ABB RAPID module: prog-1.rapid

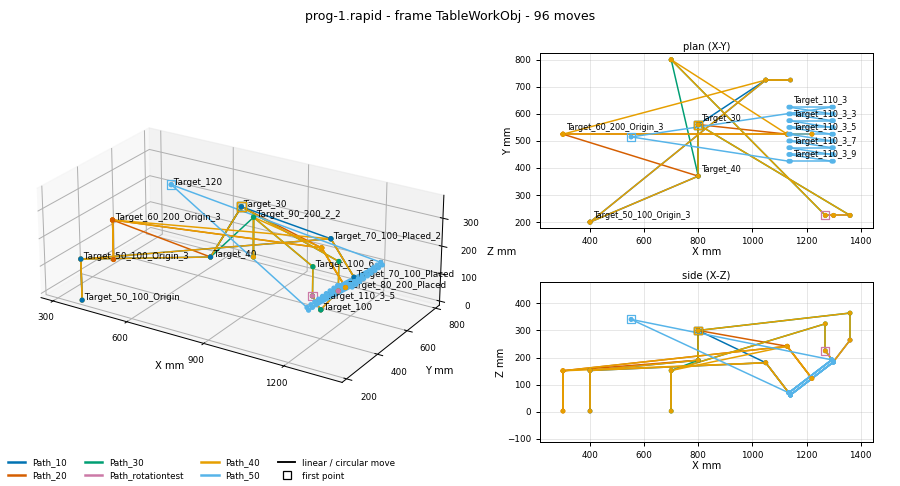
[picture p0: tool path of prog-1.rapid in frame TableWorkObj, 96 of 96 moves have a stored position in this frame; points joined in program order, loops and branches not executed]
MODULE Module1
    CONST robtarget Target_30:=[[800,560.525588833,300],[0.353553391,-0.612372436,0.612372436,0.353553391],[-1,0,-1,0],[9E+09,9E+09,9E+09,9E+09,9E+09,9E+09]];
    CONST robtarget Target_40:=[[800,370.00032529,189.999990631],[-0.000000004,-0.707106781,0.707106781,-0.000000004],[-1,0,-1,0],[9E+09,9E+09,9E+09,9E+09,9E+09,9E+09]];
    CONST robtarget Target_50_100_Origin_3:=[[400,199.9999982,152],[0.000000006,1,0,0],[0,0,-1,0],[9E+09,9E+09,9E+09,9E+09,9E+09,9E+09]];
    CONST robtarget Target_50_100_Origin:=[[400,200,2],[-0.000000006,1,0,0],[0,-1,-1,0],[9E+09,9E+09,9E+09,9E+09,9E+09,9E+09]];
    CONST robtarget Target_70_100_Placed_2:=[[1049.406562207,725,180.67251142],[-0.000000006,1,0,0],[-1,0,-2,0],[9E+09,9E+09,9E+09,9E+09,9E+09,9E+09]];
    CONST robtarget Target_70_100_Placed:=[[1140.720642254,725,61.669407321],[0,0.946930311,0,0.321438931],[-1,-1,-2,0],[9E+09,9E+09,9E+09,9E+09,9E+09,9E+09]];
    CONST robtarget Target_60_200_Origin_3:=[[300.000000926,524.99999882,151],[0.000000003,0.965925826,-0.258819045,-0.000000004],[0,0,-1,0],[9E+09,9E+09,9E+09,9E+09,9E+09,9E+09]];
    CONST robtarget Target_60_200_Origin:=[[300,525,2],[0,0.965925826,-0.258819045,0],[0,0,-1,0],[9E+09,9E+09,9E+09,9E+09,9E+09,9E+09]];
    CONST robtarget Target_80_200_Placed_2:=[[1128.741964994,525,241.548561714],[-0.000000006,1,0,0],[-1,0,-2,0],[9E+09,9E+09,9E+09,9E+09,9E+09,9E+09]];
    CONST robtarget Target_80_200_Placed:=[[1220.056045041,525,122.545460615],[0,0.946930311,0,0.321438931],[-1,-1,-2,0],[9E+09,9E+09,9E+09,9E+09,9E+09,9E+09]];
    CONST robtarget Target_90_200_2_2:=[[700,800,152],[0,0.965925826,0.258819045,0],[0,0,-2,0],[9E+09,9E+09,9E+09,9E+09,9E+09,9E+09]];
    CONST robtarget Target_90_200_2:=[[700,800,2],[0,0.965925826,0.258819045,0],[0,0,-2,0],[9E+09,9E+09,9E+09,9E+09,9E+09,9E+09]];
    CONST robtarget Target_100_6_2:=[[1269.56192856,225,324.667667022],[0.000000006,1,0,0],[-1,-1,-2,0],[9E+09,9E+09,9E+09,9E+09,9E+09,9E+09]];
    CONST robtarget Target_100_6:=[[1269.56192856,225,224.667667022],[0,0.94693013,0,0.321439465],[-1,-1,-2,0],[9E+09,9E+09,9E+09,9E+09,9E+09,9E+09]];
    CONST robtarget Target_100:=[[1300,225,185],[0,0.946930129,0,0.321439465],[-1,-1,-2,0],[9E+09,9E+09,9E+09,9E+09,9E+09,9E+09]];
    CONST robtarget Target_100_3:=[[1300,225,185],[0,0.946930129,0,-0.321439465],[-1,0,-2,0],[9E+09,9E+09,9E+09,9E+09,9E+09,9E+09]];
    CONST robtarget Target_100_3_2:=[[1360.876142881,225,264.335334045],[0,0.94693013,0,-0.321439465],[-1,0,-2,0],[9E+09,9E+09,9E+09,9E+09,9E+09,9E+09]];
    CONST robtarget Target_100_3_2_2:=[[1360.876142881,225,364.335334045],[0.000000006,1,0,0],[-1,-1,-2,0],[9E+09,9E+09,9E+09,9E+09,9E+09,9E+09]];
    CONST robtarget Target_110_2_10:=[[1293.303842438,625,191.355054252],[0.946930311,0,-0.321438931,0],[-1,-4,2,1],[9E+09,9E+09,9E+09,9E+09,9E+09,9E+09]];
    CONST robtarget Target_110_2:=[[1299.391447774,625,183.421513979],[0.946930311,0,-0.321438931,0],[-1,-4,2,1],[9E+09,9E+09,9E+09,9E+09,9E+09,9E+09]];
    CONST robtarget Target_110_3:=[[1140.720642308,625,61.669407251],[0.946930311,0,-0.321438931,0],[-1,-4,2,1],[9E+09,9E+09,9E+09,9E+09,9E+09,9E+09]];
    CONST robtarget Target_110_3_10:=[[1134.633036972,625,69.602947524],[0.946930311,0,-0.321438931,0],[-1,-4,2,1],[9E+09,9E+09,9E+09,9E+09,9E+09,9E+09]];
    CONST robtarget Target_110_2_2_2:=[[1293.303842438,600,191.355054252],[0.946930311,0,-0.321438931,0],[-1,-4,2,1],[9E+09,9E+09,9E+09,9E+09,9E+09,9E+09]];
    CONST robtarget Target_110_2_2:=[[1299.391447774,600,183.421513979],[0.946930311,0,-0.321438931,0],[-1,-4,2,1],[9E+09,9E+09,9E+09,9E+09,9E+09,9E+09]];
    CONST robtarget Target_110_3_2:=[[1140.720642308,600,61.669407251],[0.946930311,0,-0.321438931,0],[-1,-4,2,1],[9E+09,9E+09,9E+09,9E+09,9E+09,9E+09]];
    CONST robtarget Target_110_3_2_2:=[[1134.633036972,600,69.602947524],[0.946930311,0,-0.321438931,0],[-1,-4,2,1],[9E+09,9E+09,9E+09,9E+09,9E+09,9E+09]];
    CONST robtarget Target_110_2_3_2:=[[1293.303842438,575,191.355054252],[0.946930311,0,-0.321438931,0],[-1,-4,2,1],[9E+09,9E+09,9E+09,9E+09,9E+09,9E+09]];
    CONST robtarget Target_110_2_3:=[[1299.391447774,575,183.421513979],[0.946930311,0,-0.321438931,0],[-1,-4,2,1],[9E+09,9E+09,9E+09,9E+09,9E+09,9E+09]];
    CONST robtarget Target_110_3_3:=[[1140.720642308,575,61.669407251],[0.946930311,0,-0.321438931,0],[-1,-4,2,1],[9E+09,9E+09,9E+09,9E+09,9E+09,9E+09]];
    CONST robtarget Target_110_3_3_2:=[[1134.633036972,575,69.602947524],[0.946930311,0,-0.321438931,0],[-1,-4,2,1],[9E+09,9E+09,9E+09,9E+09,9E+09,9E+09]];
    CONST robtarget Target_110_2_4_2:=[[1293.303842438,550,191.355054252],[0.946930311,0,-0.321438931,0],[-1,-4,2,1],[9E+09,9E+09,9E+09,9E+09,9E+09,9E+09]];
    CONST robtarget Target_110_2_4:=[[1299.391447774,550,183.421513979],[0.946930311,0,-0.321438931,0],[-1,-4,2,1],[9E+09,9E+09,9E+09,9E+09,9E+09,9E+09]];
    CONST robtarget Target_110_3_4:=[[1140.720642308,550,61.669407251],[0.946930311,0,-0.321438931,0],[-1,-4,2,1],[9E+09,9E+09,9E+09,9E+09,9E+09,9E+09]];
    CONST robtarget Target_110_3_4_2:=[[1134.633036972,550,69.602947524],[0.946930311,0,-0.321438931,0],[-1,-4,2,1],[9E+09,9E+09,9E+09,9E+09,9E+09,9E+09]];
    CONST robtarget Target_110_2_5_2:=[[1293.303842438,525,191.355054252],[0.946930311,0,-0.321438931,0],[-1,-4,2,1],[9E+09,9E+09,9E+09,9E+09,9E+09,9E+09]];
    CONST robtarget Target_110_2_5:=[[1299.391447774,525,183.421513979],[0.946930311,0,-0.321438931,0],[-1,-4,2,1],[9E+09,9E+09,9E+09,9E+09,9E+09,9E+09]];
    CONST robtarget Target_110_3_5:=[[1140.720642308,525,61.669407251],[0.946930311,0,-0.321438931,0],[-1,-4,2,1],[9E+09,9E+09,9E+09,9E+09,9E+09,9E+09]];
    CONST robtarget Target_110_3_5_2:=[[1134.633036972,525,69.602947524],[0.946930311,0,-0.321438931,0],[-1,-4,2,1],[9E+09,9E+09,9E+09,9E+09,9E+09,9E+09]];
    CONST robtarget Target_110_2_6_2:=[[1293.303842438,500,191.355054252],[0.946930311,0,-0.321438931,0],[-1,-4,2,1],[9E+09,9E+09,9E+09,9E+09,9E+09,9E+09]];
    CONST robtarget Target_110_2_6:=[[1299.391447774,500,183.421513979],[0.946930311,0,-0.321438931,0],[-1,-4,2,1],[9E+09,9E+09,9E+09,9E+09,9E+09,9E+09]];
    CONST robtarget Target_110_3_6:=[[1140.720642308,500,61.669407251],[0.946930311,0,-0.321438931,0],[-1,-4,2,1],[9E+09,9E+09,9E+09,9E+09,9E+09,9E+09]];
    CONST robtarget Target_110_3_6_2:=[[1134.633036972,500,69.602947524],[0.946930311,0,-0.321438931,0],[-1,-4,2,1],[9E+09,9E+09,9E+09,9E+09,9E+09,9E+09]];
    CONST robtarget Target_110_2_7_2:=[[1293.303842438,475,191.355054252],[0.946930311,0,-0.321438931,0],[-1,-4,2,1],[9E+09,9E+09,9E+09,9E+09,9E+09,9E+09]];
    CONST robtarget Target_110_2_7:=[[1299.391447774,475,183.421513979],[0.946930311,0,-0.321438931,0],[-1,-4,2,1],[9E+09,9E+09,9E+09,9E+09,9E+09,9E+09]];
    CONST robtarget Target_110_3_7:=[[1140.720642308,475,61.669407251],[0.946930311,0,-0.321438931,0],[-1,-4,2,1],[9E+09,9E+09,9E+09,9E+09,9E+09,9E+09]];
    CONST robtarget Target_110_3_7_2:=[[1134.633036972,475,69.602947524],[0.946930311,0,-0.321438931,0],[-1,-4,2,1],[9E+09,9E+09,9E+09,9E+09,9E+09,9E+09]];
    CONST robtarget Target_110_2_8_2:=[[1293.303842438,450,191.355054252],[0.946930311,0,-0.321438931,0],[-1,-4,2,1],[9E+09,9E+09,9E+09,9E+09,9E+09,9E+09]];
    CONST robtarget Target_110_2_8:=[[1299.391447774,450,183.421513979],[0.946930311,0,-0.321438931,0],[-1,-4,2,1],[9E+09,9E+09,9E+09,9E+09,9E+09,9E+09]];
    CONST robtarget Target_110_3_8:=[[1140.720642308,450,61.669407251],[0.946930311,0,-0.321438931,0],[-1,-4,2,1],[9E+09,9E+09,9E+09,9E+09,9E+09,9E+09]];
    CONST robtarget Target_110_3_8_2:=[[1134.633036972,450,69.602947524],[0.946930311,0,-0.321438931,0],[-1,-4,2,1],[9E+09,9E+09,9E+09,9E+09,9E+09,9E+09]];
    CONST robtarget Target_110_2_9_2:=[[1293.303842438,425,191.355054252],[0.946930311,0,-0.321438931,0],[-1,-4,2,1],[9E+09,9E+09,9E+09,9E+09,9E+09,9E+09]];
    CONST robtarget Target_110_2_9:=[[1299.391447774,425,183.421513979],[0.946930311,0,-0.321438931,0],[-1,-4,2,1],[9E+09,9E+09,9E+09,9E+09,9E+09,9E+09]];
    CONST robtarget Target_110_3_9:=[[1140.720642308,425,61.669407251],[0.946930311,0,-0.321438931,0],[-1,-4,2,1],[9E+09,9E+09,9E+09,9E+09,9E+09,9E+09]];
    CONST robtarget Target_110_3_9_2:=[[1134.633036972,425,69.602947524],[0.946930311,0,-0.321438931,0],[-1,-4,2,1],[9E+09,9E+09,9E+09,9E+09,9E+09,9E+09]];
    CONST robtarget Target_120:=[[552,514.814,340.825],[0.612372436,0.353553391,0.612372436,0.353553391],[0,-3,2,1],[9E+09,9E+09,9E+09,9E+09,9E+09,9E+09]];
    CONST robtarget Target_Patch200:=[[300,525,2],[0,0.965925826,-0.258819045,0],[0,0,-1,0],[9E+09,9E+09,9E+09,9E+09,9E+09,9E+09]];
!***********************************************************
    !
    ! Module:  Module1
    !
    ! Description:
    !   <Insert description here>
    !
    ! Author: tgell
    !
    ! Version: 1.0
    !
    !***********************************************************


    !***********************************************************
    !
    ! Procedure main
    !
    !   This is the entry point of your program
    !
    !***********************************************************
    PROC main()
        Path_20;
        Path_50;
        !Add your code here
    ENDPROC
    PROC Path_10()
        MoveL Target_30,v400,z100,Tooldata_1\WObj:=TableWorkObj;
        MoveL Target_40,v400,z100,Tooldata_1\WObj:=TableWorkObj;
        MoveL Target_50_100_Origin_3,v400,z100,Tooldata_1\WObj:=TableWorkObj;
        MoveL Target_50_100_Origin,v60,z100,Tooldata_1\WObj:=TableWorkObj;
        WaitTime 3;
        PulseDO att_100;
        MoveL Target_50_100_Origin_3,v60,z100,Tooldata_1\WObj:=TableWorkObj;
        MoveL Target_70_100_Placed_2,v150,z100,Tooldata_1\WObj:=TableWorkObj;
        MoveL Target_70_100_Placed,v60,z100,Tooldata_1\WObj:=TableWorkObj;
        WaitTime 3;
        PulseDO det_100;
        MoveL Target_70_100_Placed_2,v60,z100,Tooldata_1\WObj:=TableWorkObj;
        MoveL Target_30,v400,z100,Tooldata_1\WObj:=TableWorkObj;
    ENDPROC
    PROC Path_20()
        MoveL Target_30,v300,z100,Tooldata_1\WObj:=TableWorkObj;
        MoveL Target_40,v300,z100,Tooldata_1\WObj:=TableWorkObj;
        MoveL Target_60_200_Origin_3,v300,z100,Tooldata_1\WObj:=TableWorkObj;
        MoveL Target_Patch200,v60,z100,Tooldata_1\WObj:=TableWorkObj;
        WaitTime 3;
        PulseDO att_200;
        MoveL Target_60_200_Origin_3,v60,z100,Tooldata_1\WObj:=TableWorkObj;
        MoveL Target_80_200_Placed_2,v100,z100,Tooldata_1\WObj:=TableWorkObj;
        MoveL Target_80_200_Placed,v60,z100,Tooldata_1\WObj:=TableWorkObj;
        WaitTime 3;
        PulseDO det_200;
        MoveL Target_80_200_Placed_2,v60,z100,Tooldata_1\WObj:=TableWorkObj;
        MoveL Target_30,v400,z100,Tooldata_1\WObj:=TableWorkObj;
        WaitTime 3;
    ENDPROC
    PROC Path_30()
        MoveL Target_30,v300,z60,Tooldata_1\WObj:=TableWorkObj;
        MoveL Target_40,v300,z60,Tooldata_1\WObj:=TableWorkObj;
        MoveL Target_90_200_2_2,v300,z60,Tooldata_1\WObj:=TableWorkObj;
        MoveL Target_90_200_2,v60,z60,Tooldata_1\WObj:=TableWorkObj;
        WaitTime 3;
        PulseDO att_200x100_L;
        PulseDO att_200x100_R;
        MoveL Target_90_200_2_2,v60,z60,Tooldata_1\WObj:=TableWorkObj;
        MoveL Target_100_6_2,v150,z60,Tooldata_1\WObj:=TableWorkObj;
        MoveL Target_100_6,v150,z60,Tooldata_1\WObj:=TableWorkObj;
        MoveL Target_100,v60,z60,Tooldata_1\WObj:=TableWorkObj;
        WaitTime 1;
        PulseDO det_200x100_L;
        MoveL Target_100_3,v5,fine,Tooldata_1\WObj:=TableWorkObj;
        WaitTime 1;
        PulseDO det_200x100_R;
        MoveL Target_100_3_2,v60,z60,Tooldata_1\WObj:=TableWorkObj;
        MoveL Target_100_3_2_2,v300,z60,Tooldata_1\WObj:=TableWorkObj;
        MoveL Target_30,v300,z60,Tooldata_1\WObj:=TableWorkObj;
    ENDPROC
    PROC Path_rotationtest()
        MoveL Target_100_6,v150,z60,Tooldata_1\WObj:=TableWorkObj;
        MoveL Target_100,v60,z60,Tooldata_1\WObj:=TableWorkObj;
        WaitTime 1;
        MoveL Target_100_3,v5,fine,Tooldata_1\WObj:=TableWorkObj;
        WaitTime 1;
        MoveL Target_100_3_2,v60,z60,Tooldata_1\WObj:=TableWorkObj;
    ENDPROC
    PROC Path_40()
        MoveL Target_30,v400,z100,Tooldata_1\WObj:=TableWorkObj;
        MoveL Target_40,v400,z100,Tooldata_1\WObj:=TableWorkObj;
        MoveL Target_50_100_Origin_3,v400,z100,Tooldata_1\WObj:=TableWorkObj;
        MoveL Target_50_100_Origin,v60,z100,Tooldata_1\WObj:=TableWorkObj;
        WaitTime 3;
        PulseDO att_100;
        MoveL Target_50_100_Origin_3,v60,z100,Tooldata_1\WObj:=TableWorkObj;
        MoveL Target_70_100_Placed_2,v150,z100,Tooldata_1\WObj:=TableWorkObj;
        MoveL Target_70_100_Placed,v60,z100,Tooldata_1\WObj:=TableWorkObj;
        WaitTime 3;
        PulseDO det_100;
        MoveL Target_70_100_Placed_2,v60,z100,Tooldata_1\WObj:=TableWorkObj;
        MoveL Target_60_200_Origin_3,v300,z100,Tooldata_1\WObj:=TableWorkObj;
        MoveL Target_Patch200,v60,z100,Tooldata_1\WObj:=TableWorkObj;
        WaitTime 3;
        PulseDO att_200;
        MoveL Target_60_200_Origin_3,v60,z100,Tooldata_1\WObj:=TableWorkObj;
        MoveL Target_80_200_Placed_2,v100,z100,Tooldata_1\WObj:=TableWorkObj;
        MoveL Target_80_200_Placed,v60,z100,Tooldata_1\WObj:=TableWorkObj;
        WaitTime 3;
        PulseDO det_200;
        MoveL Target_80_200_Placed_2,v60,z100,Tooldata_1\WObj:=TableWorkObj;
        MoveL Target_90_200_2_2,v300,z60,Tooldata_1\WObj:=TableWorkObj;
        MoveL Target_90_200_2,v60,z60,Tooldata_1\WObj:=TableWorkObj;
        WaitTime 3;
        PulseDO att_200x100_L;
        PulseDO att_200x100_R;
        MoveL Target_90_200_2_2,v60,z60,Tooldata_1\WObj:=TableWorkObj;
        MoveL Target_100_6_2,v150,z60,Tooldata_1\WObj:=TableWorkObj;
        MoveL Target_100_6,v150,z60,Tooldata_1\WObj:=TableWorkObj;
        MoveL Target_100,v60,z60,Tooldata_1\WObj:=TableWorkObj;
        WaitTime 1;
        PulseDO det_200x100_L;
        MoveL Target_100_3,v5,fine,Tooldata_1\WObj:=TableWorkObj;
        WaitTime 1;
        PulseDO det_200x100_R;
        MoveL Target_100_3_2,v60,z60,Tooldata_1\WObj:=TableWorkObj;
        MoveL Target_100_3_2_2,v300,z60,Tooldata_1\WObj:=TableWorkObj;
        MoveL Target_30,v300,z60,Tooldata_1\WObj:=TableWorkObj;
    ENDPROC
    PROC Path_50()
        MoveL Target_120,v60,z60,Tooldata_2_Roller\WObj:=TableWorkObj;
        MoveL Target_110_2_10,v150,z1,Tooldata_2_Roller\WObj:=TableWorkObj;
        MoveL Target_110_2,v150,z1,Tooldata_2_Roller\WObj:=TableWorkObj;
        MoveL Target_110_3,v150,z1,Tooldata_2_Roller\WObj:=TableWorkObj;
        MoveL Target_110_3_10,v150,z1,Tooldata_2_Roller\WObj:=TableWorkObj;
        MoveL Target_110_2_2_2,v150,z1,Tooldata_2_Roller\WObj:=TableWorkObj;
        MoveL Target_110_2_2,v150,z1,Tooldata_2_Roller\WObj:=TableWorkObj;
        MoveL Target_110_3_2,v150,z1,Tooldata_2_Roller\WObj:=TableWorkObj;
        MoveL Target_110_3_2_2,v150,z1,Tooldata_2_Roller\WObj:=TableWorkObj;
        MoveL Target_110_2_3_2,v150,z1,Tooldata_2_Roller\WObj:=TableWorkObj;
        MoveL Target_110_2_3,v150,z1,Tooldata_2_Roller\WObj:=TableWorkObj;
        MoveL Target_110_3_3,v150,z1,Tooldata_2_Roller\WObj:=TableWorkObj;
        MoveL Target_110_3_3_2,v150,z1,Tooldata_2_Roller\WObj:=TableWorkObj;
        MoveL Target_110_2_4_2,v150,z1,Tooldata_2_Roller\WObj:=TableWorkObj;
        MoveL Target_110_2_4,v150,z1,Tooldata_2_Roller\WObj:=TableWorkObj;
        MoveL Target_110_3_4,v150,z1,Tooldata_2_Roller\WObj:=TableWorkObj;
        MoveL Target_110_3_4_2,v150,z1,Tooldata_2_Roller\WObj:=TableWorkObj;
        MoveL Target_110_2_5_2,v150,z1,Tooldata_2_Roller\WObj:=TableWorkObj;
        MoveL Target_110_2_5,v150,z1,Tooldata_2_Roller\WObj:=TableWorkObj;
        MoveL Target_110_3_5,v150,z1,Tooldata_2_Roller\WObj:=TableWorkObj;
        MoveL Target_110_3_5_2,v150,z1,Tooldata_2_Roller\WObj:=TableWorkObj;
        MoveL Target_110_2_6_2,v150,z1,Tooldata_2_Roller\WObj:=TableWorkObj;
        MoveL Target_110_2_6,v150,z1,Tooldata_2_Roller\WObj:=TableWorkObj;
        MoveL Target_110_3_6,v150,z1,Tooldata_2_Roller\WObj:=TableWorkObj;
        MoveL Target_110_3_6_2,v150,z1,Tooldata_2_Roller\WObj:=TableWorkObj;
        MoveL Target_110_2_7_2,v150,z1,Tooldata_2_Roller\WObj:=TableWorkObj;
        MoveL Target_110_2_7,v150,z1,Tooldata_2_Roller\WObj:=TableWorkObj;
        MoveL Target_110_3_7,v150,z1,Tooldata_2_Roller\WObj:=TableWorkObj;
        MoveL Target_110_3_7_2,v150,z1,Tooldata_2_Roller\WObj:=TableWorkObj;
        MoveL Target_110_2_8_2,v150,z1,Tooldata_2_Roller\WObj:=TableWorkObj;
        MoveL Target_110_2_8,v150,z1,Tooldata_2_Roller\WObj:=TableWorkObj;
        MoveL Target_110_3_8,v150,z1,Tooldata_2_Roller\WObj:=TableWorkObj;
        MoveL Target_110_3_8_2,v150,z1,Tooldata_2_Roller\WObj:=TableWorkObj;
        MoveL Target_110_2_9_2,v150,z1,Tooldata_2_Roller\WObj:=TableWorkObj;
        MoveL Target_110_2_9,v150,z1,Tooldata_2_Roller\WObj:=TableWorkObj;
        MoveL Target_110_3_9,v150,z1,Tooldata_2_Roller\WObj:=TableWorkObj;
        MoveL Target_110_3_9_2,v150,z1,Tooldata_2_Roller\WObj:=TableWorkObj;
        MoveL Target_120,v60,z60,Tooldata_2_Roller\WObj:=TableWorkObj;
    ENDPROC
ENDMODULE
